(* Logix 5000 project; controller Safety vendor 1 type 14 code 86 rev 19.11; software revision 19.01; part 4 of 17 *)
(* tags used below, declared in another part *)
   A1_IO : UDT_CardSts[32];   // A1 Point I/O
   A1_IOSts_Flt : BOOL;   // A1 Point IO Module Fault ( 1= Faulted)
   A1_S20_ModFlt : ALIAS FOR Flt_Modules[0].0;   // A1 Point I/O Slot20 Module Fault (1 = Fault)
   A1_S21_ModFlt : ALIAS FOR Flt_Modules[0].1;   // A1 Point I/O Slot21 Module Fault (1 = Fault)
   C1_IO : UDT_CardSts[32];   // C1 Point I/O
   C1_IOSts_Flt : BOOL;   // C1 Point IO Module Fault ( 1= Faulted)
   C1_S12_ModFlt : ALIAS FOR Flt_Modules[0].2;   // C1 Point I/O Slot12 Module Fault (1 = Fault)
   ChgMe : BOOL;
   CHPLC_IO : UDT_CardSts[32];   // CHPLC Point I/O
   CHPLC_IOSts_Flt : BOOL;   // CHPLC Point IO Module Fault ( 1= Faulted)
   CHPLC_S1_ModFlt : ALIAS FOR Flt_Modules[0].3;   // CHPLC Point I/O Slot01 Module Fault (1 = Fault)
   CHPLC_S2_ModFlt : ALIAS FOR Flt_Modules[0].4;   // CHPLC Point I/O Slot02 Module Fault (1 = Fault)
   CHPLC_S3_ModFlt : ALIAS FOR Flt_Modules[0].5;   // CHPLC Point I/O Slot03 Module Fault (1 = Fault)
   CHPLC_S4_ModFlt : ALIAS FOR Flt_Modules[0].6;   // CHPLC Point I/O Slot04 Module Fault (1 = Fault)
   CHPLC_S5_ModFlt : ALIAS FOR Flt_Modules[0].7;   // CHPLC Point I/O Slot05 Module Fault (1 = Fault)
   CHPLC_S6_ModFlt : ALIAS FOR Flt_Modules[0].8;   // CHPLC Point I/O Slot06 Module Fault (1 = Fault)
   CommCards_OK : DINT;   // Comm Cards OK
   D1_IO : UDT_CardSts[32];   // D1 Point I/O
   D1_IOSts_Flt : BOOL;   // D1 Point IO Module Fault ( 1= Faulted)
   D1_S12_ModFlt : ALIAS FOR Flt_Modules[0].9;   // D1 Point I/O Slot12 Module Fault (1 = Fault)
   DPD_IO : UDT_CardSts[32];   // DPD Point I/O
   DPD_IOSts_Flt : BOOL;   // DPD Point IO Module Fault ( 1= Faulted)
   DPD_S14_ModFlt : ALIAS FOR Flt_Modules[0].10;   // DPD Point I/O Slot14 Module Fault (1 = Fault)
   DPD_S15_ModFlt : ALIAS FOR Flt_Modules[0].11;   // DPD Point I/O Slot15 Module Fault (1 = Fault)
   E1_IO : UDT_CardSts[32];   // E1 Point I/O
   E1_IOSts_Flt : BOOL;   // E1 Point IO Module Fault ( 1= Faulted)
   E1_S10_ModFlt : ALIAS FOR Flt_Modules[0].12;   // E1 Point I/O Slot10 Module Fault (1 = Fault)
   ES_IndJog_PB : BOOL;   // Exit Section Individual Jog Select ( 1= Req Individual)
   ES_Line_JogPB : BOOL;   // Exit Section Line Jog PB ( 1= Ind Jog )
   ES_Line_RunPB : BOOL;   // Exit Section Line Run PB ( 1= Run)
   ES_Line_StopPB : BOOL;   // Exit Section Line Stop PB ( 1= OK) (0=Stop)
   ES_Line_ThreadPB : BOOL;   // Exit Section Line Thread PB ( 1= Thread)
   ES_TndJog_PB : BOOL;   // Exit Section Tandem Jog PB (1= Tandem Jog Sel)
   ESTOP_x201PB040_Flt : ALIAS FOR Flt_Estops.0;   // OS1 Line EStop Pushbutton Fault ( 1= Fault)
   ESTOP_x211PB040_Flt : ALIAS FOR Flt_Estops.1;   // OS2 Line EStop Pushbutton Fault ( 1= Fault)
   ESTOP_x221PB040_Flt : ALIAS FOR Flt_Estops.2;   // OS3 Line EStop Pushbutton Fault ( 1= Fault)
   ESTOP_x231PB040_Flt : ALIAS FOR Flt_Estops.3;   // OS4N Line EStop Pushbutton Fault ( 1= Fault)
   ESTOP_x241PB040_Flt : ALIAS FOR Flt_Estops.4;   // OS4S Line EStop Pushbutton Fault ( 1= Fault)
   ESTOP_x251PB040_Flt : ALIAS FOR Flt_Estops.5;   // OS5 Line EStop Pushbutton Fault ( 1= Fault)
   ESTOP_x261PB040_Flt : ALIAS FOR Flt_Estops.6;   // OS6 Line EStop Pushbutton Fault ( 1= Fault)
   ESTOP_x271PB040_Flt : ALIAS FOR Flt_Estops.7;   // OS8 Line EStop Pushbutton Fault ( 1= Fault)
   ESTOP_x281PB040_Flt : ALIAS FOR Flt_Estops.8;   // OS9 Line EStop Pushbutton Fault ( 1= Fault)
   ESTOP_x291PB040_Flt : ALIAS FOR Flt_Estops.9;   // OS11 Line EStop Pushbutton Fault ( 1= Fault)
   ESTOP_x301PB040_Flt : ALIAS FOR Flt_Estops.10;   // OS13 Line EStop Pushbutton Fault ( 1= Fault)
   ESTOP_x311PB040_Flt : ALIAS FOR Flt_Estops.11;   // OS14 Line EStop Pushbutton Fault ( 1= Fault)
   ESTOP_x311PB130_Flt : ALIAS FOR Flt_Estops.17;   // OS14 Shear EStop Pushbutton Fault ( 1= Fault)
   ESTOP_x321PB040_Flt : ALIAS FOR Flt_Estops.12;   // OS15 Line EStop Pushbutton Fault ( 1= Fault)
   ESTOP_x331PB040_Flt : ALIAS FOR Flt_Estops.13;   // OS16 Line EStop Pushbutton Fault ( 1= Fault)
   ESTOP_x480PB470_Flt : ALIAS FOR Flt_Estops.14;   // DPD Line EStop Pushbutton Fault ( 1= Fault)
   ESTOP_x480PB550_Flt : ALIAS FOR Flt_Estops.15;   // DPD Line EStop Pushbutton Fault ( 1= Fault)
   ESTOP_x519LS470_Flt : ALIAS FOR Flt_Estops.18;   // G1 Line EStop Tripwire Limit Switch Fault ( 1= Fault)
   ESTOP_x533PB470_Flt : ALIAS FOR Flt_Estops.16;   // H1 Line EStop Pushbutton Fault ( 1= Fault)
   ExConHydPump_AutoStart : BOOL;   // (From Mach) Exit Conveyor Hydraulic Pump Auto Start Command
   F1_IO : UDT_CardSts[32];   // F1 Point I/O
   F1_IOSts_Flt : BOOL;   // F1 Point IO Module Fault ( 1= Faulted)
   F1_S19_ModFlt : ALIAS FOR Flt_Modules[0].13;   // F1 Point I/O Slot19 Module Fault (1 = Fault)
   F1_S20_ModFlt : ALIAS FOR Flt_Modules[0].14;   // F1 Point I/O Slot20 Module Fault (1 = Fault)
   Flt_Estops : DINT;   // Estop Fault Word
   Flt_Modules : DINT[5];   // Point IO Module Fault Word
   Flt_SafeOff : DINT[3];   // Safe Off Fault Word
   Flt_Starter : DINT;   // Starter Fault Word
   FltsToCitect : DINT[64];   // Faults to Citect
   FromCitect : DINT[64];   // (From Citect)
   FromMach : DINT[35];   // (FromMach)
   FromMachine : DINT[35];   // (FromMach)
   FromShearDie : DINT[35];   // (From Shear Die)
   FVR_y702MTR191_Flt : ALIAS FOR Flt_Starter.4;   // Rewind Pinch Roll Starter Fault ( 1= Fault)
   FVR_y708MTR080_Flt : ALIAS FOR Flt_Starter.1;   // Flattener Drive Motor Starter Fault ( 1= Fault)
   FVR_y708MTR250_Flt : ALIAS FOR Flt_Starter.0;   // Unwind Hold Down Roll Starter Fault ( 1= Fault)
   FVR_y753MTR190_Flt : ALIAS FOR Flt_Starter.2;   // Trimmer Pinch Roll Starter Fault ( 1= Fault)
   FVR_y761MTR081_Flt : ALIAS FOR Flt_Starter.3;   // Trimmer Scrap Conveyor Starter Fault ( 1= Fault)
   FVR_y778MTR080_Flt : ALIAS FOR Flt_Starter.5;   // Shear Die Crank Starter Fault ( 1= Fault)
   FVR_y802MTR080_Flt : ALIAS FOR Flt_Starter.6;   // Stacker Side Guide Lift Starter Fault ( 1= Fault)
   FVR_y802MTR230_Flt : ALIAS FOR Flt_Starter.8;   // Scrap Horizontal Conveyor Starter Fault ( 1= Fault)
   FVR_y802MTR231_Flt : ALIAS FOR Flt_Starter.7;   // Stacker Chain Conveyor Starter Fault ( 1= Fault)
   G1_IO : UDT_CardSts[32];   // G1 Point I/O
   G1_IOSts_Flt : BOOL;   // G1 Point IO Module Fault ( 1= Faulted)
   G1_S11_ModFlt : ALIAS FOR Flt_Modules[0].15;   // G1 Point I/O Slot11 Module Fault (1 = Fault)
   G1_S12_ModFlt : ALIAS FOR Flt_Modules[0].16;   // G1 Point I/O Slot12 Module Fault (1 = Fault)
   H1_IO : UDT_CardSts[32];   // H1 Point I/O
   H1_IOSts_Flt : BOOL;   // H1 Point IO Module Fault ( 1= Faulted)
   H1_S5_ModFlt : ALIAS FOR Flt_Modules[0].17;   // H1 Point I/O Slot05 Module Fault (1 = Fault)
   H1_S6_ModFlt : ALIAS FOR Flt_Modules[0].18;   // H1 Point I/O Slot06 Module Fault (1 = Fault)
   HydPumps_AutoStart : BOOL;   // (From Mach) Hydraulic Pumps Auto Start Active
   IOCards_OK : DINT;   // Point I/O Cards OK
   Local_ModFlts : DINT;   // Local Card Fault Status
   LubePumps_AutoStart : BOOL;   // (From Mach) Lube Pumps Auto Start Active
   Machine_HB_Flt : BOOL;   // Machine Heartbeat Fault ( 1= Fault)
   MCC1_IO : UDT_CardSts[32];   // MCC1 Point I/O
   MCC1_IOSts_Flt : BOOL;   // MCC1 Point IO Module Fault ( 1= Faulted)
   MCC1_S1_ModFlt : ALIAS FOR Flt_Modules[2].0;   // MCC1 Point I/O Slot01 Module Fault (1 = Fault)
   MCC1_S6_ModFlt : ALIAS FOR Flt_Modules[2].1;   // MCC1 Point I/O Slot06 Module Fault (1 = Fault)
   MCC2_IO : UDT_CardSts[32];   // MCC2 Point I/O
   MCC2_IOSts_Flt : BOOL;   // MCC2 Point IO Module Fault ( 1= Faulted)
   MCC2_S1_ModFlt : ALIAS FOR Flt_Modules[2].2;   // MCC2 Point I/O Slot01 Module Fault (1 = Fault)
   MCC2_S2_ModFlt : ALIAS FOR Flt_Modules[2].3;   // MCC2 Point I/O Slot02 Module Fault (1 = Fault)
   MCC3_IO : UDT_CardSts[32];   // MCC3 Point I/O
   MCC3_IOSts_Flt : BOOL;   // MCC3 Point IO Module Fault ( 1= Faulted)
   MCC3_S1_ModFlt : ALIAS FOR Flt_Modules[2].4;   // MCC3 Point I/O Slot01 Module Fault (1 = Fault)
   MCC3_S3_ModFlt : ALIAS FOR Flt_Modules[2].5;   // MCC3 Point I/O Slot03 Module Fault (1 = Fault)
   MCC3_S4_ModFlt : ALIAS FOR Flt_Modules[2].6;   // MCC3 Point I/O Slot04 Module Fault (1 = Fault)
   MCC4_IO : UDT_CardSts[32];   // MCC4 Point I/O
   MCC4_IOSts_Flt : BOOL;   // MCC-4 Point IO Module Fault ( 1= Faulted)
   MCC4_S1_ModFlt : ALIAS FOR Flt_Modules[2].7;   // MCC4 Point I/O Slot01 Module Fault (1 = Fault)
   MCC4_S3_ModFlt : ALIAS FOR Flt_Modules[2].8;   // MCC4 Point I/O Slot03 Module Fault (1 = Fault)
   MCC4_S4_ModFlt : ALIAS FOR Flt_Modules[2].9;   // MCC4 Point I/O Slot04 Module Fault (1 = Fault)
   MCC5_IO : UDT_CardSts[32];   // MCC5 Point I/O
   MCC5_IOSts_Flt : BOOL;   // MCC-5 Point IO Module Fault ( 1= Faulted)
   MCC5_S1_ModFlt : ALIAS FOR Flt_Modules[2].10;   // MCC5 Point I/O Slot01 Module Fault (1 = Fault)
   MCC5_S3_ModFlt : ALIAS FOR Flt_Modules[2].11;   // MCC5 Point I/O Slot03 Module Fault (1 = Fault)
   MCC5_S4_ModFlt : ALIAS FOR Flt_Modules[2].12;   // MCC5 Point I/O Slot04 Module Fault (1 = Fault)
   MCC5_S5_ModFlt : ALIAS FOR Flt_Modules[2].13;   // MCC5 Point I/O Slot05 Module Fault (1 = Fault)
   OS11_IO : UDT_CardSts[32];   // OS11 Point I/O
   OS11_IOSts_Flt : BOOL;   // OS11 Point IO Module Fault ( 1= Faulted)
   OS11_S1_ModFlt : ALIAS FOR Flt_Modules[1].11;   // OS11 Point I/O Slot01 Module Fault (1 = Fault)
   OS13_IO : UDT_CardSts[32];   // OS13 Point I/O
   OS13_IOSts_Flt : BOOL;   // OS13 Point IO Module Fault ( 1= Faulted)
   OS13_S1_ModFlt : ALIAS FOR Flt_Modules[1].12;   // OS13 Point I/O Slot01 Module Fault (1 = Fault)
   OS14_IO : UDT_CardSts[32];   // OS14 Point I/O
   OS14_IOSts_Flt : BOOL;   // OS14 Point IO Module Fault ( 1= Faulted)
   OS14_S1_ModFlt : ALIAS FOR Flt_Modules[1].13;   // OS14 Point I/O Slot01 Module Fault (1 = Fault)
   OS15_IO : UDT_CardSts[32];   // OS15 Point I/O
   OS15_IOSts_Flt : BOOL;   // OS15 Point IO Module Fault ( 1= Faulted)
   OS15_S1_ModFlt : ALIAS FOR Flt_Modules[1].14;   // OS15 Point I/O Slot01 Module Fault (1 = Fault)
   OS16_IO : UDT_CardSts[32];   // OS16 Point I/O
   OS16_IOSts_Flt : BOOL;   // OS16 Point IO Module Fault ( 1= Faulted)
   OS16_S1_ModFlt : ALIAS FOR Flt_Modules[1].15;   // OS16 Point I/O Slot01 Module Fault (1 = Fault)
   OS1_IO : UDT_CardSts[32];   // OS1 Point I/O
   OS1_IOSts_Flt : BOOL;   // OS1 Point IO Module Fault ( 1= Faulted)
   OS1_S1_ModFlt : ALIAS FOR Flt_Modules[1].0;   // OS1 Point I/O Slot01 Module Fault (1 = Fault)
   OS2_IO : UDT_CardSts[32];   // OS2 Point I/O
   OS2_IOSts_Flt : BOOL;   // OS2 Point IO Module Fault ( 1= Faulted)
   OS2_S1_ModFlt : ALIAS FOR Flt_Modules[1].1;   // OS2 Point I/O Slot01 Module Fault (1 = Fault)
   OS3_IO : UDT_CardSts[32];   // OS3 Point I/O
   OS3_IOSts_Flt : BOOL;   // OS3 Point IO Module Fault ( 1= Faulted)
   OS3_S1_ModFlt : ALIAS FOR Flt_Modules[1].2;   // OS3 Point I/O Slot01 Module Fault (1 = Fault)
   OS4N_IO : UDT_CardSts[32];   // OS4N Point I/O
   OS4N_IOSts_Flt : BOOL;   // OS4N Point IO Module Fault ( 1= Faulted)
   OS4N_S1_ModFlt : ALIAS FOR Flt_Modules[1].3;   // OS4N Point I/O Slot01 Module Fault (1 = Fault)
   OS4N_S5_ModFlt : ALIAS FOR Flt_Modules[1].4;   // OS4N Point I/O Slot05 Module Fault (1 = Fault)
   OS4S_IO : UDT_CardSts[32];   // OS4S Point I/O
   OS4S_IOSts_Flt : BOOL;   // OS4S Point IO Module Fault ( 1= Faulted)
   OS4S_S1_ModFlt : ALIAS FOR Flt_Modules[1].5;   // OS4S Point I/O Slot01 Module Fault (1 = Fault)
   OS4S_S5_ModFlt : ALIAS FOR Flt_Modules[1].6;   // OS4S Point I/O Slot05 Module Fault (1 = Fault)
   OS5_IO : UDT_CardSts[32];   // OS5 Point I/O
   OS5_IOSts_Flt : BOOL;   // OS5 Point IO Module Fault ( 1= Faulted)
   OS5_S1_ModFlt : ALIAS FOR Flt_Modules[1].7;   // OS5 Point I/O Slot01 Module Fault (1 = Fault)
   OS6_IO : UDT_CardSts[32];   // OS6 Point I/O
   OS6_IOSts_Flt : BOOL;   // OS6 Point IO Module Fault ( 1= Faulted)
   OS6_S1_ModFlt : ALIAS FOR Flt_Modules[1].8;   // OS6 Point I/O Slot01 Module Fault (1 = Fault)
   OS8_IO : UDT_CardSts[32];   // OS8 Point I/O
   OS8_IOSts_Flt : BOOL;   // OS8 Point IO Module Fault ( 1= Faulted)
   OS8_S1_ModFlt : ALIAS FOR Flt_Modules[1].9;   // OS8 Point I/O Slot01 Module Fault (1 = Fault)
   OS9_IO : UDT_CardSts[32];   // OS9 Point I/O
   OS9_IOSts_Flt : BOOL;   // OS9 Point IO Module Fault ( 1= Faulted)
   OS9_S1_ModFlt : ALIAS FOR Flt_Modules[1].10;   // OS9 Point I/O Slot01 Module Fault (1 = Fault)
   Rem_ModFlts : DINT;   // Remote IO Comm Faults
   SafeOff_y172CR460_Flt : ALIAS FOR Flt_SafeOff[0].0;   // Shear Die Main Contactor Relay Fault ( 1= Fault)
   SafeOff_y172CR510_Flt : ALIAS FOR Flt_SafeOff[0].1;   // Shear Die Drive Enable Relay Fault ( 1= Fault)
   SafeOff_y613CR460_Flt : ALIAS FOR Flt_SafeOff[0].2;   // Unwind Op Side Main Contactor Relay Fault ( 1= Fault)
   SafeOff_y613CR510_Flt : ALIAS FOR Flt_SafeOff[0].3;   // Unwind Op Side Drive Enable Relay Fault ( 1= Fault)
   SafeOff_y613CR550_Flt : ALIAS FOR Flt_SafeOff[0].4;   // Unwind Drive Side Main Contactor Relay Fault ( 1= Fault)
   SafeOff_y613CR590_Flt : ALIAS FOR Flt_SafeOff[0].5;   // Unwind Drive Side Drive Enable Relay Fault ( 1= Fault)
   SafeOff_y613CR630_Flt : ALIAS FOR Flt_SafeOff[0].6;   // #1 Entry Bridle Roll 2 Main Contactor Relay Fault ( 1= Fault)
   SafeOff_y613CR670_Flt : ALIAS FOR Flt_SafeOff[0].7;   // #1 Entry Bridle Roll 2 Drive Enable Relay Fault ( 1= Fault)
   SafeOff_y613CR710_Flt : ALIAS FOR Flt_SafeOff[0].8;   // #2 Entry Bridle Roll 3 Main Contactor Relay Fault ( 1= Fault)
   SafeOff_y613CR750_Flt : ALIAS FOR Flt_SafeOff[0].9;   // #2 Entry Bridle Roll 3 Drive Enable Relay Fault ( 1= Fault)
   SafeOff_y614CR040_Flt : ALIAS FOR Flt_SafeOff[0].10;   // #1 Exit Bridle Roll 6 Main Contactor Relay Fault ( 1= Fault)
   SafeOff_y614CR090_Flt : ALIAS FOR Flt_SafeOff[0].11;   // #1 Exit Bridle Roll 6 Drive Enable Relay Fault ( 1= Fault)
   SafeOff_y614CR130_Flt : ALIAS FOR Flt_SafeOff[0].12;   // #2 Exit Bridle Roll 7 Main Contactor Relay Fault ( 1= Fault)
   SafeOff_y614CR170_Flt : ALIAS FOR Flt_SafeOff[0].13;   // #2 Exit Bridle Roll 7 Drive Enable Relay Fault ( 1= Fault)
   SafeOff_y614CR210_Flt : ALIAS FOR Flt_SafeOff[0].14;   // Rewind Main Contactor Relay Fault ( 1= Fault)
   SafeOff_y614CR250_Flt : ALIAS FOR Flt_SafeOff[0].15;   // Rewind Drive Enable Relay Fault ( 1= Fault)
   ScrapModeOn : BOOL;   // Scrap Mode Selected ( 1= Requested)
   SDPLC_IO : UDT_CardSts[32];   // SDPLC Point I/O
   SDPLC_IOSts_Flt : BOOL;   // SDPLC Point IO Module Fault ( 1= Faulted)
   SDPLC_S1_ModFlt : ALIAS FOR Flt_Modules[0].19;   // SDPLC Point I/O Slot01 Module Fault (1 = Fault)
   SDPLC_S2_ModFlt : ALIAS FOR Flt_Modules[0].20;   // SDPLC Point I/O Slot02 Module Fault (1 = Fault)
   Shear_HB_Flt : BOOL;   // Shear Heartbeat Fault ( 1= Fault)
   SrPRLubePump_AutoStart : BOOL;   // (From Mach) Shear Pinch Roll Lube Pump Auto Start Command
   StHydPump_AutoStart : BOOL;   // (From Mach) Sheeter Hydraulic Pump Auto Start Command
   StPRLubePump_AutoStart : BOOL;   // (From Mach) Sheeter Pinch Roll Lube Pump Auto Start Command
   Sy_ClrFlt : BOOL;   // System Clear Fault
   VS2_IO : UDT_CardSts[32];   // VS2 Point I/O
   VS2_IOSts_Flt : BOOL;   // VS2 Point IO Module Fault ( 1= Faulted)
   VS2_S10_ModFlt : ALIAS FOR Flt_Modules[0].21;   // VS2 Point I/O Slot10 Module Fault (1 = Fault)
   x301SS540a : BOOL;   // Sheeter Pinch Roll Jog Forward SS
   x301SS540b : BOOL;   // Sheeter Pinch Roll Jog Reverse SS
   x312PB700 : BOOL;   // Product Conveyor Jog Forward PB
   x312PB740 : BOOL;   // Product Conveyor Jog Reverse PB
   x312SS460a : BOOL;   // Scrap Conveyor Jog Forward SS
   x312SS460b : BOOL;   // Scrap Conveyor Jog Reverse SS
   x313SS460a : BOOL;   // Shear Conveyor Jog Forward SS
   x313SS460b : BOOL;   // Shear Conveyor Jog Reverse SS
   x314SS040a : BOOL;   // Shear Pinch Roll Jog Forward SS
   x314SS040b : BOOL;   // Shear Pinch Roll Jog Reverse SS
   x315SS040a : BOOL;   // Sheeter Pinch Roll Jog Forward SS
   x315SS040b : BOOL;   // Sheeter Pinch Roll Jog Reverse SS
   x775MTR280RF : BOOL;   // (From Shear DIe) Shear Pinch Roll Lube Run Fdbk
   x781MTR080RF : BOOL;   // (From Shear DIe) Sheeter Pinch Roll Lube Run Fdbk
   x781MTR190RF : BOOL;   // (From Shear DIe) Sheeter Hyd Pump Run Fdbk
   x813MTR080RF : BOOL;   // (From Shear DIe) Exit Conveyor Hyd Pump Run Fdbk
(* CardSts, continued *)

ROUTINE Remote_IO   (* ladder *)
// Remote IO Card Status
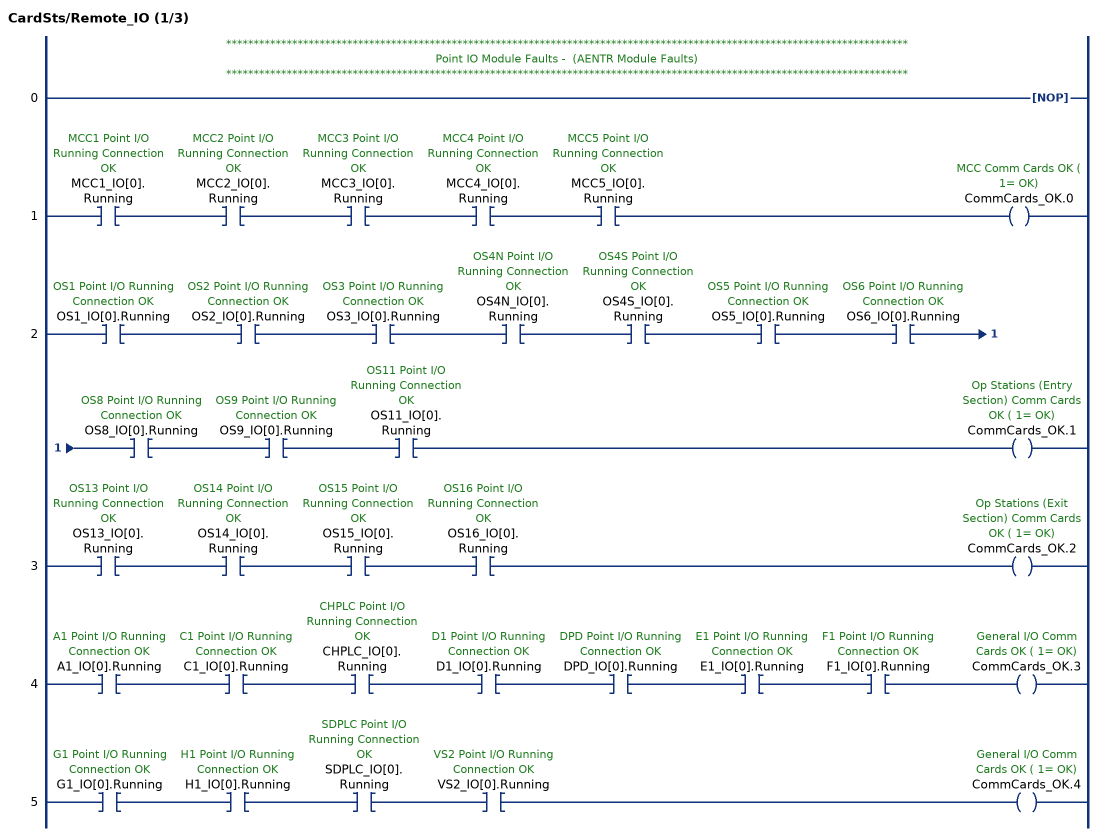
   // ****************************************************************************************************************************
   // Point IO Module Faults -  (AENTR Module Faults)
   // ****************************************************************************************************************************
   0: NOP();
   1: XIC(MCC1_IO[0].Running)XIC(MCC2_IO[0].Running)XIC(MCC3_IO[0].Running)XIC(MCC4_IO[0].Running)XIC(MCC5_IO[0].Running)OTE(CommCards_OK.0);
   2: XIC(OS1_IO[0].Running)XIC(OS2_IO[0].Running)XIC(OS3_IO[0].Running)XIC(OS4N_IO[0].Running)XIC(OS4S_IO[0].Running)XIC(OS5_IO[0].Running)XIC(OS6_IO[0].Running)XIC(OS8_IO[0].Running)XIC(OS9_IO[0].Running)XIC(OS11_IO[0].Running)OTE(CommCards_OK.1);
   3: XIC(OS13_IO[0].Running)XIC(OS14_IO[0].Running)XIC(OS15_IO[0].Running)XIC(OS16_IO[0].Running)OTE(CommCards_OK.2);
   4: XIC(A1_IO[0].Running)XIC(C1_IO[0].Running)XIC(CHPLC_IO[0].Running)XIC(D1_IO[0].Running)XIC(DPD_IO[0].Running)XIC(E1_IO[0].Running)XIC(F1_IO[0].Running)OTE(CommCards_OK.3);
   5: XIC(G1_IO[0].Running)XIC(H1_IO[0].Running)XIC(SDPLC_IO[0].Running)XIC(VS2_IO[0].Running)OTE(CommCards_OK.4);
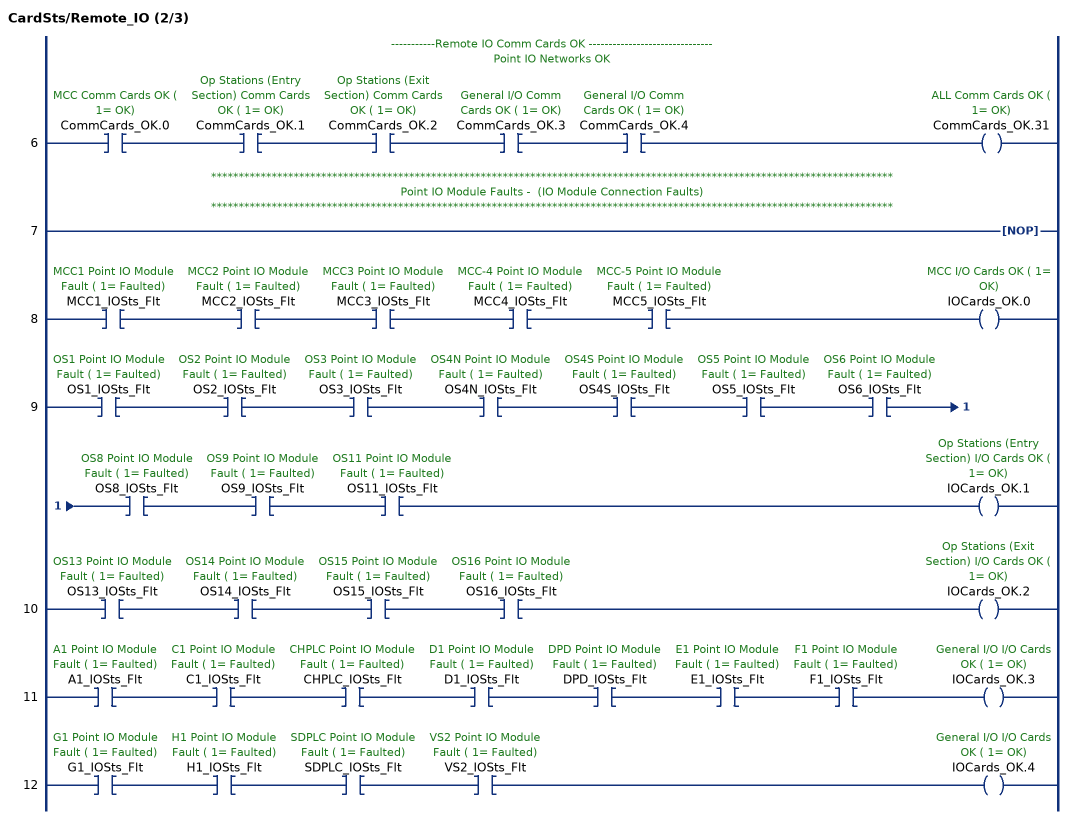
   // -----------Remote IO Comm Cards OK -------------------------------
   // Point IO Networks OK
   6: XIC(CommCards_OK.0)XIC(CommCards_OK.1)XIC(CommCards_OK.2)XIC(CommCards_OK.3)XIC(CommCards_OK.4)OTE(CommCards_OK.31);
   // ****************************************************************************************************************************
   // Point IO Module Faults -  (IO Module Connection Faults)
   // ****************************************************************************************************************************
   7: NOP();
   8: XIC(MCC1_IOSts_Flt)XIC(MCC2_IOSts_Flt)XIC(MCC3_IOSts_Flt)XIC(MCC4_IOSts_Flt)XIC(MCC5_IOSts_Flt)OTE(IOCards_OK.0);
   9: XIC(OS1_IOSts_Flt)XIC(OS2_IOSts_Flt)XIC(OS3_IOSts_Flt)XIC(OS4N_IOSts_Flt)XIC(OS4S_IOSts_Flt)XIC(OS5_IOSts_Flt)XIC(OS6_IOSts_Flt)XIC(OS8_IOSts_Flt)XIC(OS9_IOSts_Flt)XIC(OS11_IOSts_Flt)OTE(IOCards_OK.1);
   10: XIC(OS13_IOSts_Flt)XIC(OS14_IOSts_Flt)XIC(OS15_IOSts_Flt)XIC(OS16_IOSts_Flt)OTE(IOCards_OK.2);
   11: XIC(A1_IOSts_Flt)XIC(C1_IOSts_Flt)XIC(CHPLC_IOSts_Flt)XIC(D1_IOSts_Flt)XIC(DPD_IOSts_Flt)XIC(E1_IOSts_Flt)XIC(F1_IOSts_Flt)OTE(IOCards_OK.3);
   12: XIC(G1_IOSts_Flt)XIC(H1_IOSts_Flt)XIC(SDPLC_IOSts_Flt)XIC(VS2_IOSts_Flt)OTE(IOCards_OK.4);
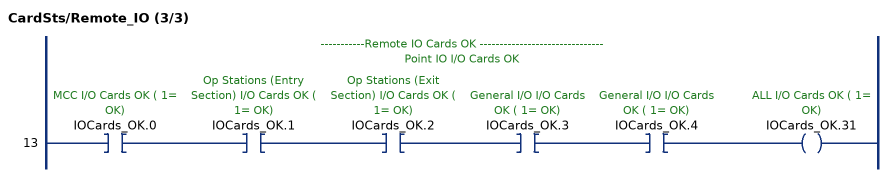
   // -----------Remote IO Cards OK -------------------------------
   // Point IO I/O Cards OK
   13: XIC(IOCards_OK.0)XIC(IOCards_OK.1)XIC(IOCards_OK.2)XIC(IOCards_OK.3)XIC(IOCards_OK.4)OTE(IOCards_OK.31);
END_ROUTINE

ROUTINE SDPLC_IO   (* ladder *)
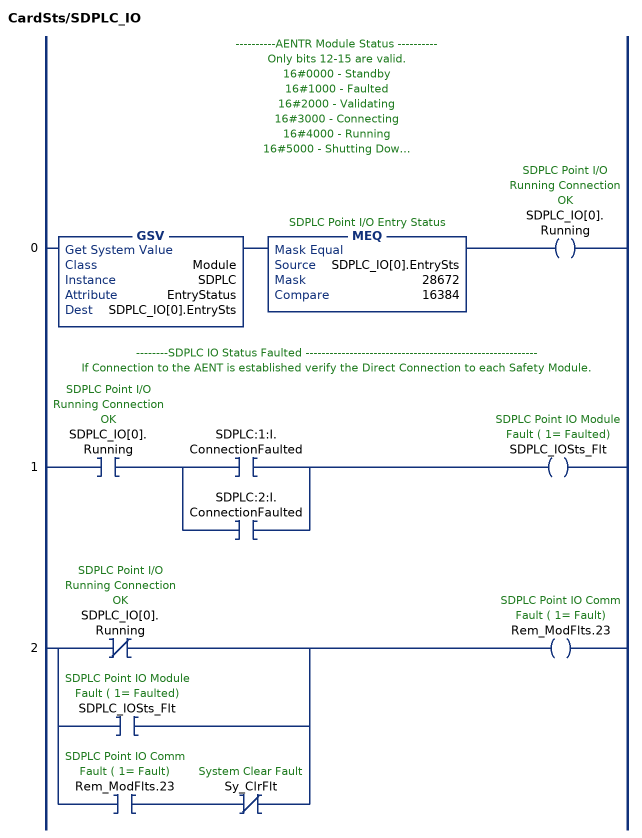
   // ----------AENTR Module Status ----------
   // Only bits 12-15 are valid.
   // 16#0000 - Standby
   // 16#1000 - Faulted
   // 16#2000 - Validating
   // 16#3000 - Connecting
   // 16#4000 - Running
   // 16#5000 - Shutting Down
   // 16#6000 - Inhibited
   // 16#7000 - Waiting
   0: GSV(Module,SDPLC,EntryStatus,SDPLC_IO[0].EntrySts)MEQ(SDPLC_IO[0].EntrySts,28672,16384)OTE(SDPLC_IO[0].Running);
   // --------SDPLC IO Status Faulted ----------------------------------------------------------
   // If Connection to the AENT is established verify the Direct Connection to each Safety Module.
   1: XIC(SDPLC_IO[0].Running)[XIC(SDPLC:1:I.ConnectionFaulted) ,XIC(SDPLC:2:I.ConnectionFaulted) ]OTE(SDPLC_IOSts_Flt);
   2: [XIO(SDPLC_IO[0].Running) ,XIC(SDPLC_IOSts_Flt) ,XIC(Rem_ModFlts.23) XIO(Sy_ClrFlt) ]OTE(Rem_ModFlts.23);
END_ROUTINE

ROUTINE VS2_IO   (* ladder *)
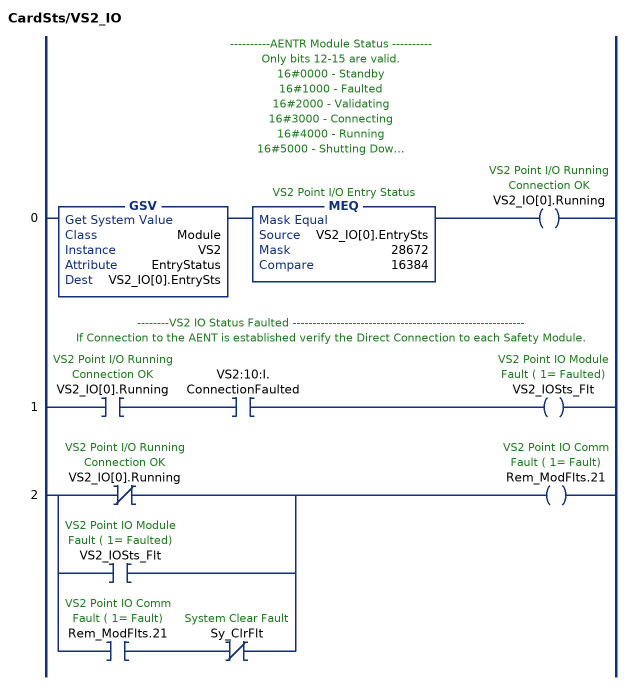
   // ----------AENTR Module Status ----------
   // Only bits 12-15 are valid.
   // 16#0000 - Standby
   // 16#1000 - Faulted
   // 16#2000 - Validating
   // 16#3000 - Connecting
   // 16#4000 - Running
   // 16#5000 - Shutting Down
   // 16#6000 - Inhibited
   // 16#7000 - Waiting
   0: GSV(Module,VS2,EntryStatus,VS2_IO[0].EntrySts)MEQ(VS2_IO[0].EntrySts,28672,16384)OTE(VS2_IO[0].Running);
   // --------VS2 IO Status Faulted ----------------------------------------------------------
   // If Connection to the AENT is established verify the Direct Connection to each Safety Module.
   1: XIC(VS2_IO[0].Running)XIC(VS2:10:I.ConnectionFaulted)OTE(VS2_IOSts_Flt);
   2: [XIO(VS2_IO[0].Running) ,XIC(VS2_IOSts_Flt) ,XIC(Rem_ModFlts.21) XIO(Sy_ClrFlt) ]OTE(Rem_ModFlts.21);
END_ROUTINE
END_PROGRAM

PROGRAM Comms   (* main routine MainRoutine *)
// Communications to Others

ROUTINE FltsToCitect   (* ladder *)
// Faults to the
// Citect System
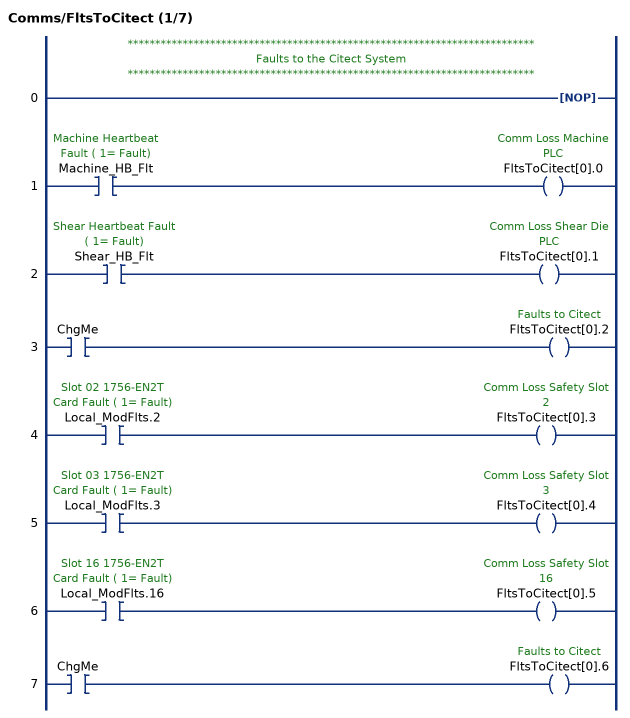
   // **************************************************************************
   // Faults to the Citect System
   // **************************************************************************
   0: NOP();
   1: XIC(Machine_HB_Flt)OTE(FltsToCitect[0].0);
   2: XIC(Shear_HB_Flt)OTE(FltsToCitect[0].1);
   3: XIC(ChgMe)OTE(FltsToCitect[0].2);
   4: XIC(Local_ModFlts.2)OTE(FltsToCitect[0].3);
   5: XIC(Local_ModFlts.3)OTE(FltsToCitect[0].4);
   6: XIC(Local_ModFlts.16)OTE(FltsToCitect[0].5);
   7: XIC(ChgMe)OTE(FltsToCitect[0].6);
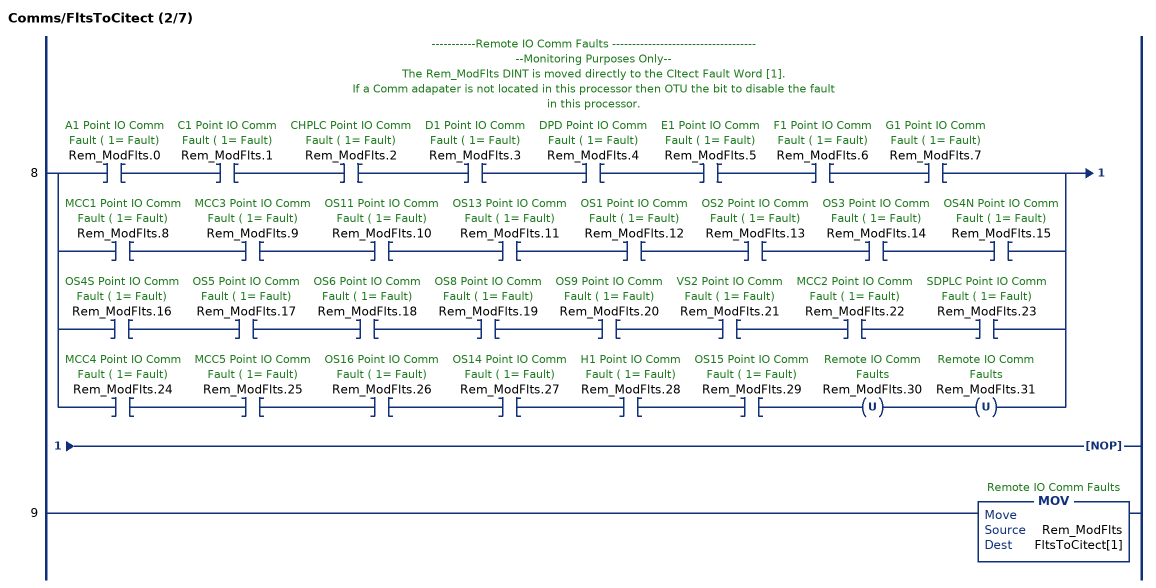
   // -----------Remote IO Comm Faults ------------------------------------
   // --Monitoring Purposes Only--
   // The Rem_ModFlts DINT is moved directly to the CItect Fault Word [1].
   // If a Comm adapater is not located in this processor then OTU the bit to disable the fault
   // in this processor.
   8: [XIC(Rem_ModFlts.0) XIC(Rem_ModFlts.1) XIC(Rem_ModFlts.2) XIC(Rem_ModFlts.3) XIC(Rem_ModFlts.4) XIC(Rem_ModFlts.5) XIC(Rem_ModFlts.6) XIC(Rem_ModFlts.7) ,XIC(Rem_ModFlts.8) XIC(Rem_ModFlts.9) XIC(Rem_ModFlts.10) XIC(Rem_ModFlts.11) XIC(Rem_ModFlts.12) XIC(Rem_ModFlts.13) XIC(Rem_ModFlts.14) XIC(Rem_ModFlts.15) ,XIC(Rem_ModFlts.16) XIC(Rem_ModFlts.17) XIC(Rem_ModFlts.18) XIC(Rem_ModFlts.19) XIC(Rem_ModFlts.20) XIC(Rem_ModFlts.21) XIC(Rem_ModFlts.22) XIC(Rem_ModFlts.23) ,XIC(Rem_ModFlts.24) XIC(Rem_ModFlts.25) XIC(Rem_ModFlts.26) XIC(Rem_ModFlts.27) XIC(Rem_ModFlts.28) XIC(Rem_ModFlts.29) OTU(Rem_ModFlts.30) OTU(Rem_ModFlts.31) ]NOP();
   9: MOV(Rem_ModFlts,FltsToCitect[1]);
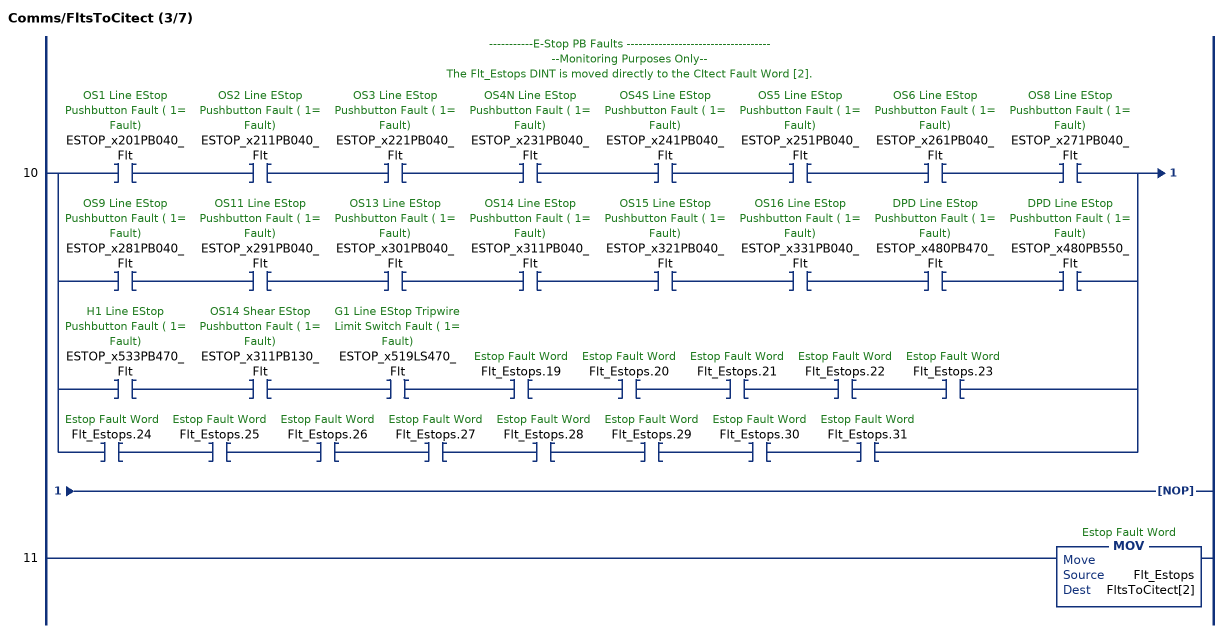
   // -----------E-Stop PB Faults ------------------------------------
   // --Monitoring Purposes Only--
   // The Flt_Estops DINT is moved directly to the CItect Fault Word [2].
   10: [XIC(ESTOP_x201PB040_Flt) XIC(ESTOP_x211PB040_Flt) XIC(ESTOP_x221PB040_Flt) XIC(ESTOP_x231PB040_Flt) XIC(ESTOP_x241PB040_Flt) XIC(ESTOP_x251PB040_Flt) XIC(ESTOP_x261PB040_Flt) XIC(ESTOP_x271PB040_Flt) ,XIC(ESTOP_x281PB040_Flt) XIC(ESTOP_x291PB040_Flt) XIC(ESTOP_x301PB040_Flt) XIC(ESTOP_x311PB040_Flt) XIC(ESTOP_x321PB040_Flt) XIC(ESTOP_x331PB040_Flt) XIC(ESTOP_x480PB470_Flt) XIC(ESTOP_x480PB550_Flt) ,XIC(ESTOP_x533PB470_Flt) XIC(ESTOP_x311PB130_Flt) XIC(ESTOP_x519LS470_Flt) XIC(Flt_Estops.19) XIC(Flt_Estops.20) XIC(Flt_Estops.21) XIC(Flt_Estops.22) XIC(Flt_Estops.23) ,XIC(Flt_Estops.24) XIC(Flt_Estops.25) XIC(Flt_Estops.26) XIC(Flt_Estops.27) XIC(Flt_Estops.28) XIC(Flt_Estops.29) XIC(Flt_Estops.30) XIC(Flt_Estops.31) ]NOP();
   11: MOV(Flt_Estops,FltsToCitect[2]);
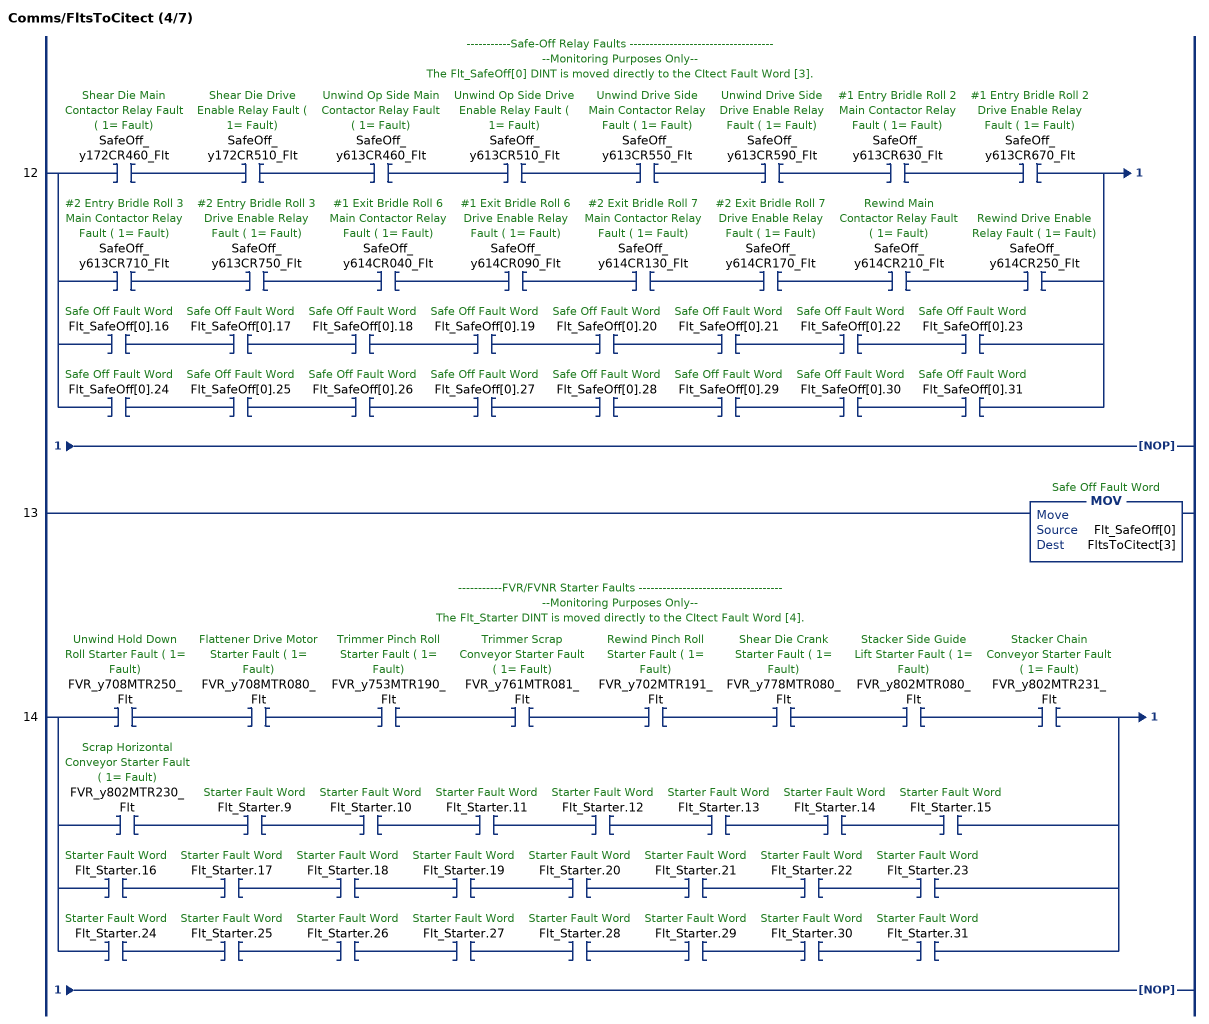
   // -----------Safe-Off Relay Faults ------------------------------------
   // --Monitoring Purposes Only--
   // The Flt_SafeOff[0] DINT is moved directly to the CItect Fault Word [3].
   12: [XIC(SafeOff_y172CR460_Flt) XIC(SafeOff_y172CR510_Flt) XIC(SafeOff_y613CR460_Flt) XIC(SafeOff_y613CR510_Flt) XIC(SafeOff_y613CR550_Flt) XIC(SafeOff_y613CR590_Flt) XIC(SafeOff_y613CR630_Flt) XIC(SafeOff_y613CR670_Flt) ,XIC(SafeOff_y613CR710_Flt) XIC(SafeOff_y613CR750_Flt) XIC(SafeOff_y614CR040_Flt) XIC(SafeOff_y614CR090_Flt) XIC(SafeOff_y614CR130_Flt) XIC(SafeOff_y614CR170_Flt) XIC(SafeOff_y614CR210_Flt) XIC(SafeOff_y614CR250_Flt) ,XIC(Flt_SafeOff[0].16) XIC(Flt_SafeOff[0].17) XIC(Flt_SafeOff[0].18) XIC(Flt_SafeOff[0].19) XIC(Flt_SafeOff[0].20) XIC(Flt_SafeOff[0].21) XIC(Flt_SafeOff[0].22) XIC(Flt_SafeOff[0].23) ,XIC(Flt_SafeOff[0].24) XIC(Flt_SafeOff[0].25) XIC(Flt_SafeOff[0].26) XIC(Flt_SafeOff[0].27) XIC(Flt_SafeOff[0].28) XIC(Flt_SafeOff[0].29) XIC(Flt_SafeOff[0].30) XIC(Flt_SafeOff[0].31) ]NOP();
   13: MOV(Flt_SafeOff[0],FltsToCitect[3]);
   // -----------FVR/FVNR Starter Faults ------------------------------------
   // --Monitoring Purposes Only--
   // The Flt_Starter DINT is moved directly to the CItect Fault Word [4].
   14: [XIC(FVR_y708MTR250_Flt) XIC(FVR_y708MTR080_Flt) XIC(FVR_y753MTR190_Flt) XIC(FVR_y761MTR081_Flt) XIC(FVR_y702MTR191_Flt) XIC(FVR_y778MTR080_Flt) XIC(FVR_y802MTR080_Flt) XIC(FVR_y802MTR231_Flt) ,XIC(FVR_y802MTR230_Flt) XIC(Flt_Starter.9) XIC(Flt_Starter.10) XIC(Flt_Starter.11) XIC(Flt_Starter.12) XIC(Flt_Starter.13) XIC(Flt_Starter.14) XIC(Flt_Starter.15) ,XIC(Flt_Starter.16) XIC(Flt_Starter.17) XIC(Flt_Starter.18) XIC(Flt_Starter.19) XIC(Flt_Starter.20) XIC(Flt_Starter.21) XIC(Flt_Starter.22) XIC(Flt_Starter.23) ,XIC(Flt_Starter.24) XIC(Flt_Starter.25) XIC(Flt_Starter.26) XIC(Flt_Starter.27) XIC(Flt_Starter.28) XIC(Flt_Starter.29) XIC(Flt_Starter.30) XIC(Flt_Starter.31) ]NOP();
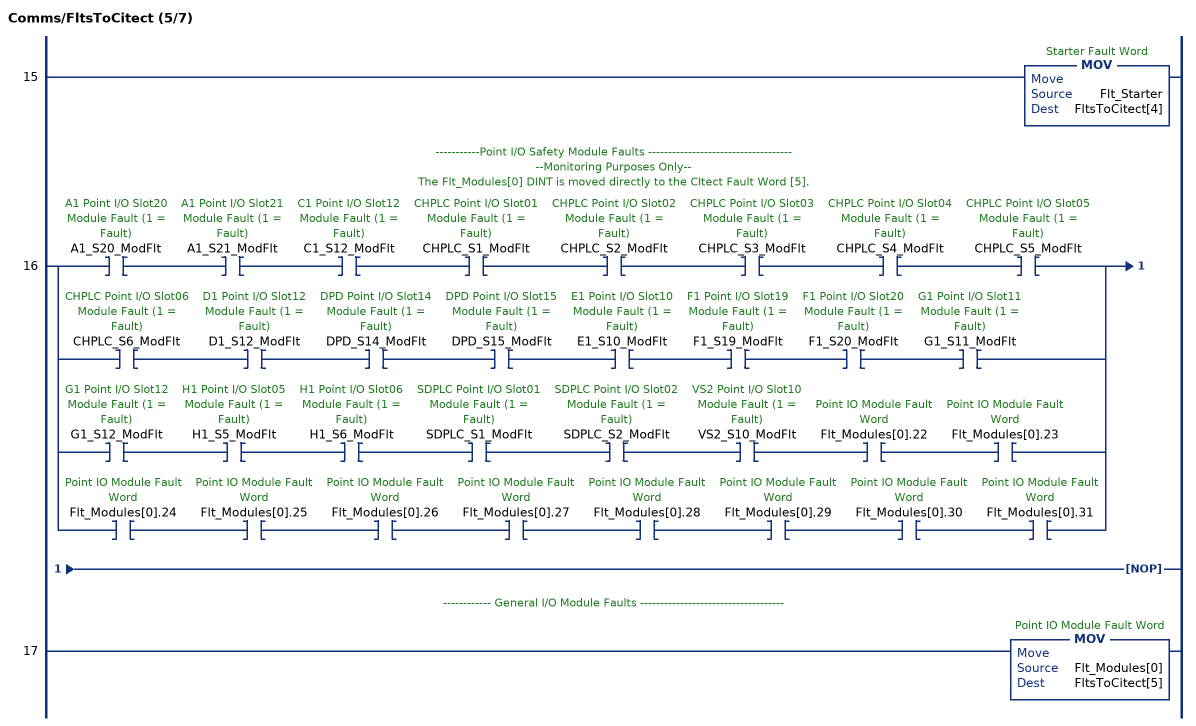
   15: MOV(Flt_Starter,FltsToCitect[4]);
   // -----------Point I/O Safety Module Faults ------------------------------------
   // --Monitoring Purposes Only--
   // The Flt_Modules[0] DINT is moved directly to the CItect Fault Word [5].
   16: [XIC(A1_S20_ModFlt) XIC(A1_S21_ModFlt) XIC(C1_S12_ModFlt) XIC(CHPLC_S1_ModFlt) XIC(CHPLC_S2_ModFlt) XIC(CHPLC_S3_ModFlt) XIC(CHPLC_S4_ModFlt) XIC(CHPLC_S5_ModFlt) ,XIC(CHPLC_S6_ModFlt) XIC(D1_S12_ModFlt) XIC(DPD_S14_ModFlt) XIC(DPD_S15_ModFlt) XIC(E1_S10_ModFlt) XIC(F1_S19_ModFlt) XIC(F1_S20_ModFlt) XIC(G1_S11_ModFlt) ,XIC(G1_S12_ModFlt) XIC(H1_S5_ModFlt) XIC(H1_S6_ModFlt) XIC(SDPLC_S1_ModFlt) XIC(SDPLC_S2_ModFlt) XIC(VS2_S10_ModFlt) XIC(Flt_Modules[0].22) XIC(Flt_Modules[0].23) ,XIC(Flt_Modules[0].24) XIC(Flt_Modules[0].25) XIC(Flt_Modules[0].26) XIC(Flt_Modules[0].27) XIC(Flt_Modules[0].28) XIC(Flt_Modules[0].29) XIC(Flt_Modules[0].30) XIC(Flt_Modules[0].31) ]NOP();
   // ------------ General I/O Module Faults ------------------------------------
   17: MOV(Flt_Modules[0],FltsToCitect[5]);
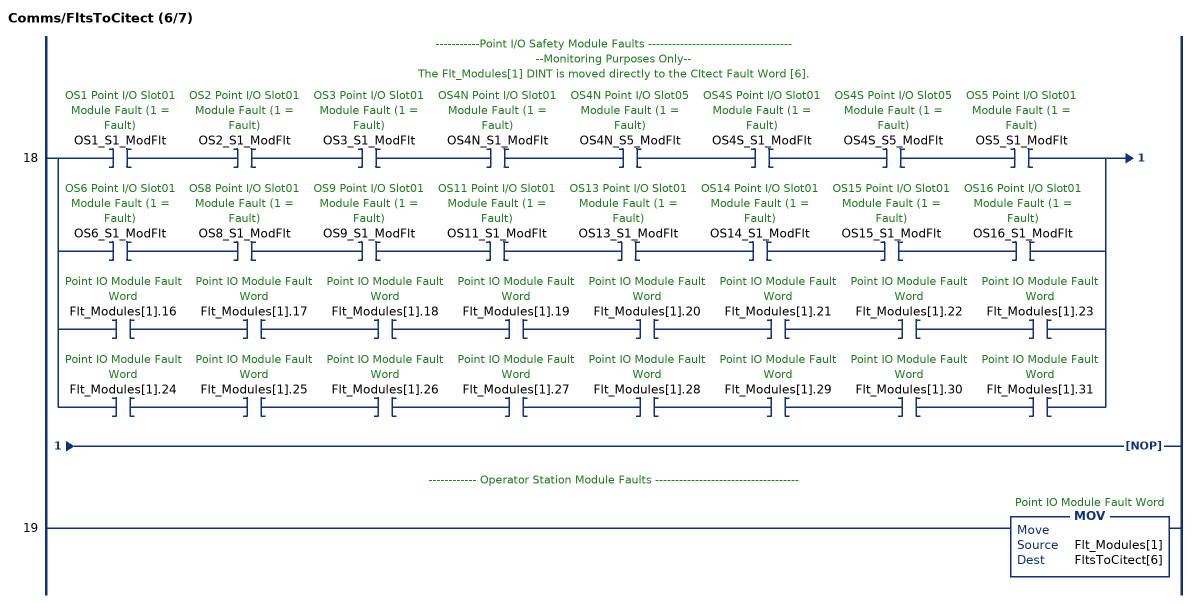
   // -----------Point I/O Safety Module Faults ------------------------------------
   // --Monitoring Purposes Only--
   // The Flt_Modules[1] DINT is moved directly to the CItect Fault Word [6].
   18: [XIC(OS1_S1_ModFlt) XIC(OS2_S1_ModFlt) XIC(OS3_S1_ModFlt) XIC(OS4N_S1_ModFlt) XIC(OS4N_S5_ModFlt) XIC(OS4S_S1_ModFlt) XIC(OS4S_S5_ModFlt) XIC(OS5_S1_ModFlt) ,XIC(OS6_S1_ModFlt) XIC(OS8_S1_ModFlt) XIC(OS9_S1_ModFlt) XIC(OS11_S1_ModFlt) XIC(OS13_S1_ModFlt) XIC(OS14_S1_ModFlt) XIC(OS15_S1_ModFlt) XIC(OS16_S1_ModFlt) ,XIC(Flt_Modules[1].16) XIC(Flt_Modules[1].17) XIC(Flt_Modules[1].18) XIC(Flt_Modules[1].19) XIC(Flt_Modules[1].20) XIC(Flt_Modules[1].21) XIC(Flt_Modules[1].22) XIC(Flt_Modules[1].23) ,XIC(Flt_Modules[1].24) XIC(Flt_Modules[1].25) XIC(Flt_Modules[1].26) XIC(Flt_Modules[1].27) XIC(Flt_Modules[1].28) XIC(Flt_Modules[1].29) XIC(Flt_Modules[1].30) XIC(Flt_Modules[1].31) ]NOP();
   // ------------ Operator Station Module Faults ------------------------------------
   19: MOV(Flt_Modules[1],FltsToCitect[6]);
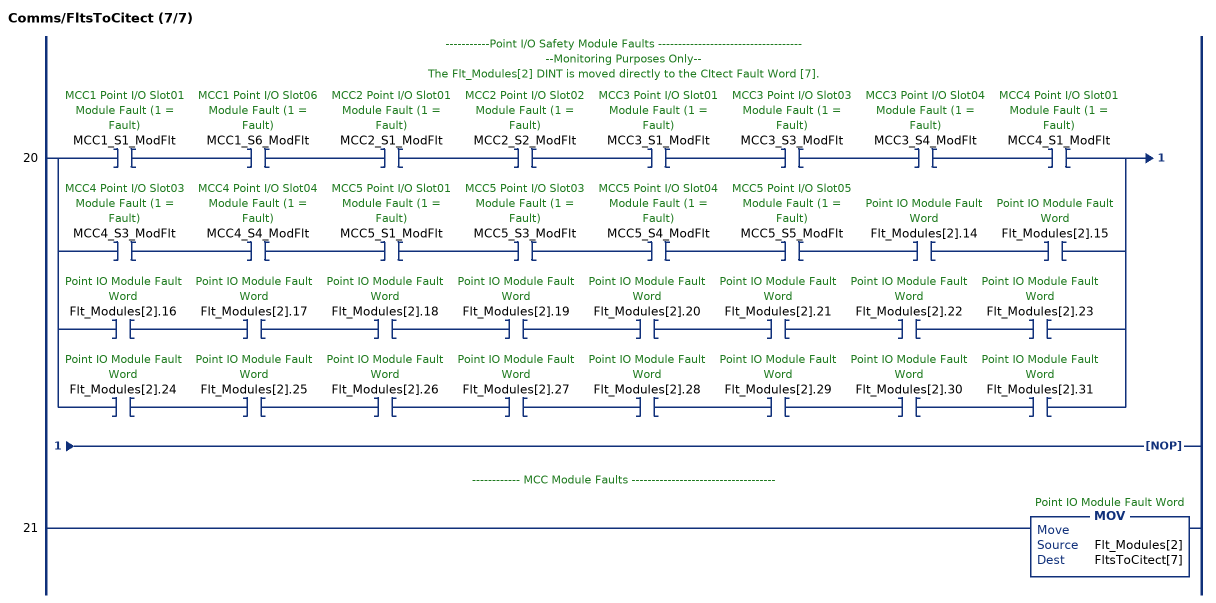
   // -----------Point I/O Safety Module Faults ------------------------------------
   // --Monitoring Purposes Only--
   // The Flt_Modules[2] DINT is moved directly to the CItect Fault Word [7].
   20: [XIC(MCC1_S1_ModFlt) XIC(MCC1_S6_ModFlt) XIC(MCC2_S1_ModFlt) XIC(MCC2_S2_ModFlt) XIC(MCC3_S1_ModFlt) XIC(MCC3_S3_ModFlt) XIC(MCC3_S4_ModFlt) XIC(MCC4_S1_ModFlt) ,XIC(MCC4_S3_ModFlt) XIC(MCC4_S4_ModFlt) XIC(MCC5_S1_ModFlt) XIC(MCC5_S3_ModFlt) XIC(MCC5_S4_ModFlt) XIC(MCC5_S5_ModFlt) XIC(Flt_Modules[2].14) XIC(Flt_Modules[2].15) ,XIC(Flt_Modules[2].16) XIC(Flt_Modules[2].17) XIC(Flt_Modules[2].18) XIC(Flt_Modules[2].19) XIC(Flt_Modules[2].20) XIC(Flt_Modules[2].21) XIC(Flt_Modules[2].22) XIC(Flt_Modules[2].23) ,XIC(Flt_Modules[2].24) XIC(Flt_Modules[2].25) XIC(Flt_Modules[2].26) XIC(Flt_Modules[2].27) XIC(Flt_Modules[2].28) XIC(Flt_Modules[2].29) XIC(Flt_Modules[2].30) XIC(Flt_Modules[2].31) ]NOP();
   // ------------ MCC Module Faults ------------------------------------
   21: MOV(Flt_Modules[2],FltsToCitect[7]);
END_ROUTINE

ROUTINE FromCitect   (* ladder *)
// Signals
// From Citect System
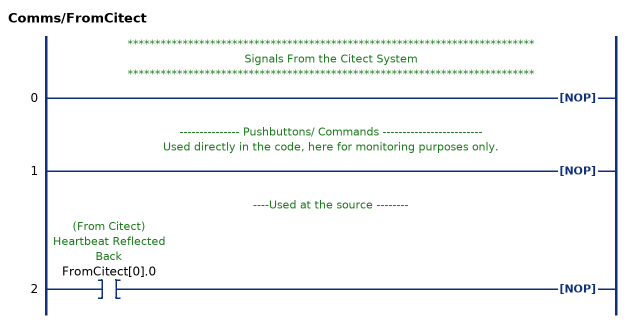
   // **************************************************************************
   // Signals From the Citect System
   // **************************************************************************
   0: NOP();
   // --------------- Pushbuttons/ Commands -------------------------
   // Used directly in the code, here for monitoring purposes only.
   1: NOP();
   // ----Used at the source --------
   2: XIC(FromCitect[0].0)NOP();
END_ROUTINE

ROUTINE FromMach   (* ladder *)
// Signals
// from Machine Processor
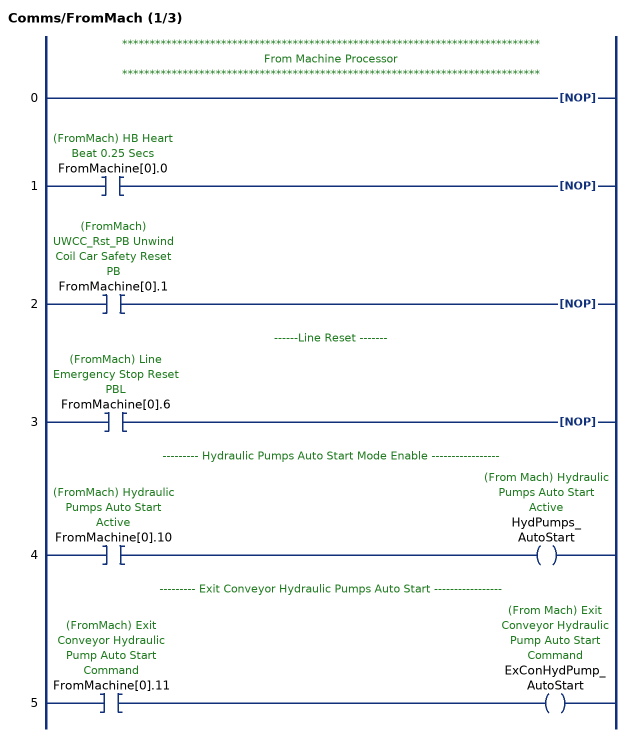
   // ****************************************************************************
   // From Machine Processor
   // ****************************************************************************
   0: NOP();
   1: XIC(FromMachine[0].0)NOP();
   2: XIC(FromMachine[0].1)NOP();
   // ------Line Reset -------
   3: XIC(FromMachine[0].6)NOP();
   // --------- Hydraulic Pumps Auto Start Mode Enable -----------------
   4: XIC(FromMachine[0].10)OTE(HydPumps_AutoStart);
   // --------- Exit Conveyor Hydraulic Pumps Auto Start -----------------
   5: XIC(FromMachine[0].11)OTE(ExConHydPump_AutoStart);
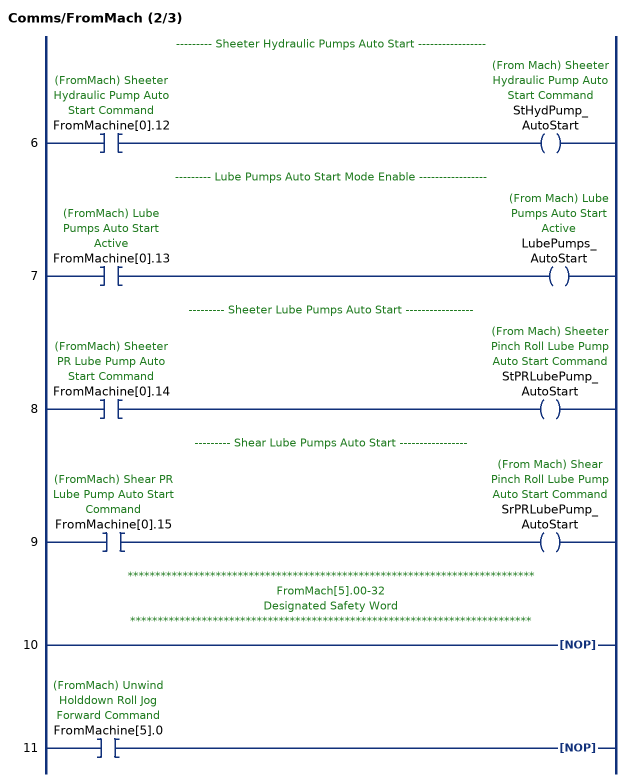
   // --------- Sheeter Hydraulic Pumps Auto Start -----------------
   6: XIC(FromMachine[0].12)OTE(StHydPump_AutoStart);
   // --------- Lube Pumps Auto Start Mode Enable -----------------
   7: XIC(FromMachine[0].13)OTE(LubePumps_AutoStart);
   // --------- Sheeter Lube Pumps Auto Start -----------------
   8: XIC(FromMachine[0].14)OTE(StPRLubePump_AutoStart);
   // --------- Shear Lube Pumps Auto Start -----------------
   9: XIC(FromMachine[0].15)OTE(SrPRLubePump_AutoStart);
   // **************************************************************************
   // FromMach[5].00-32
   // Designated Safety Word
   // *************************************************************************
   10: NOP();
   11: XIC(FromMachine[5].0)NOP();
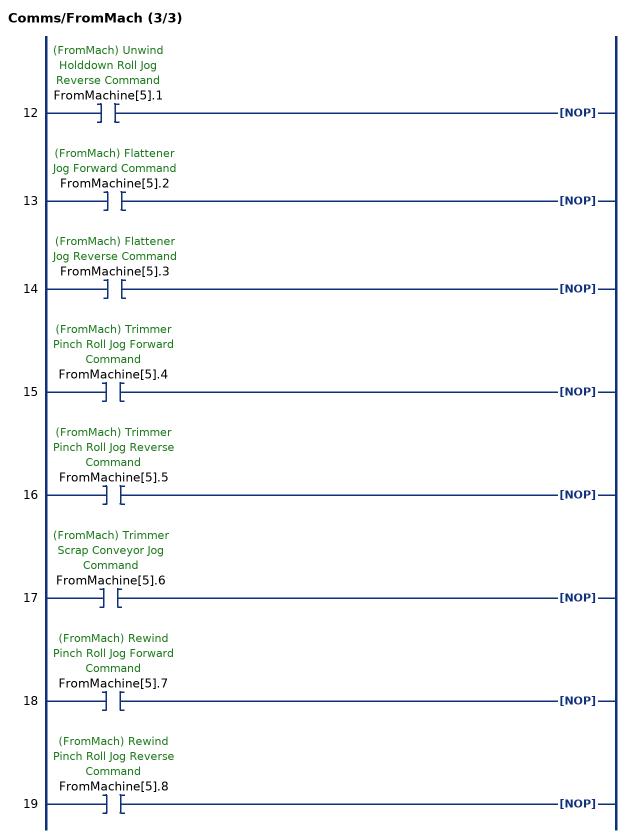
   12: XIC(FromMachine[5].1)NOP();
   13: XIC(FromMachine[5].2)NOP();
   14: XIC(FromMachine[5].3)NOP();
   15: XIC(FromMachine[5].4)NOP();
   16: XIC(FromMachine[5].5)NOP();
   17: XIC(FromMachine[5].6)NOP();
   18: XIC(FromMachine[5].7)NOP();
   19: XIC(FromMachine[5].8)NOP();
END_ROUTINE

ROUTINE FromShDie   (* ladder *)
// Signals
// from Shear Die Processor
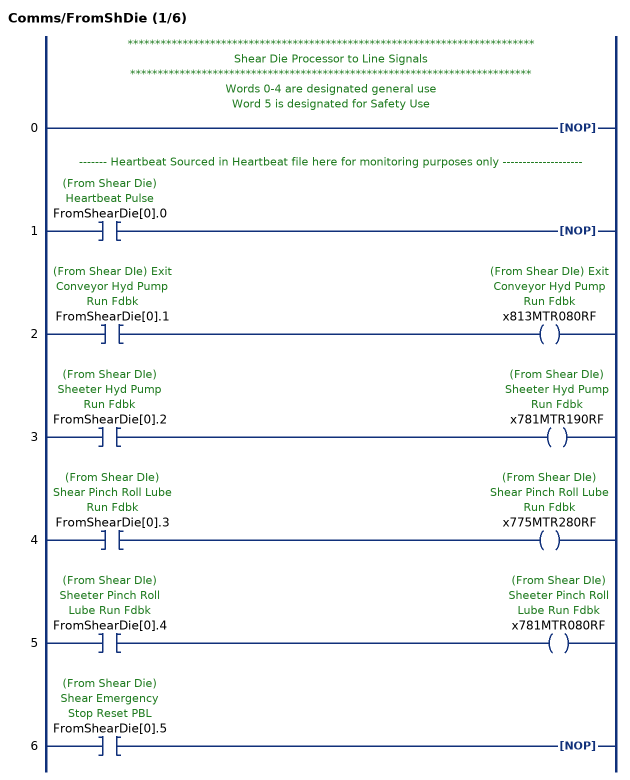
   // **************************************************************************
   // Shear Die Processor to Line Signals
   // *************************************************************************
   // Words 0-4 are designated general use
   // Word 5 is designated for Safety Use
   0: NOP();
   // ------- Heartbeat Sourced in Heartbeat file here for monitoring purposes only --------------------
   1: XIC(FromShearDie[0].0)NOP();
   2: XIC(FromShearDie[0].1)OTE(x813MTR080RF);
   3: XIC(FromShearDie[0].2)OTE(x781MTR190RF);
   4: XIC(FromShearDie[0].3)OTE(x775MTR280RF);
   5: XIC(FromShearDie[0].4)OTE(x781MTR080RF);
   6: XIC(FromShearDie[0].5)NOP();
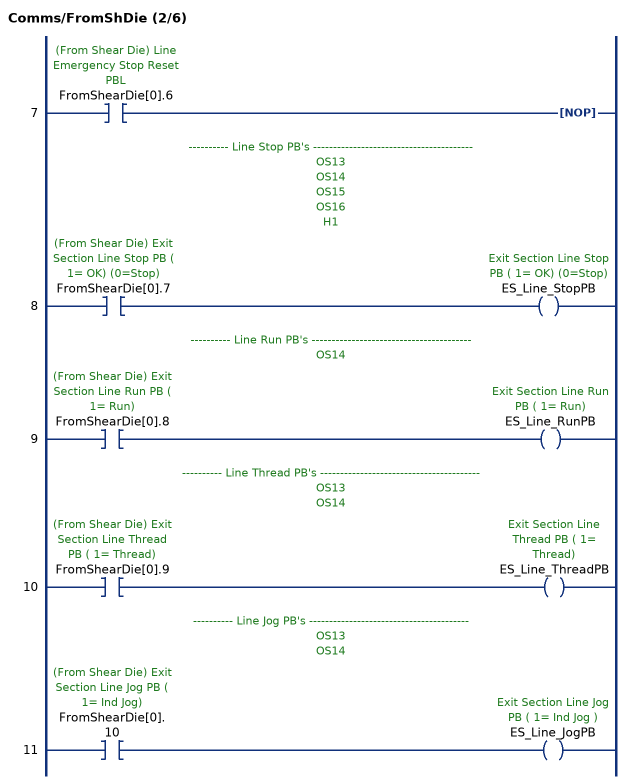
   7: XIC(FromShearDie[0].6)NOP();
   // ---------- Line Stop PB's ----------------------------------------
   // OS13
   // OS14
   // OS15
   // OS16
   // H1
   8: XIC(FromShearDie[0].7)OTE(ES_Line_StopPB);
   // ---------- Line Run PB's ----------------------------------------
   // OS14
   9: XIC(FromShearDie[0].8)OTE(ES_Line_RunPB);
   // ---------- Line Thread PB's ----------------------------------------
   // OS13
   // OS14
   10: XIC(FromShearDie[0].9)OTE(ES_Line_ThreadPB);
   // ---------- Line Jog PB's ----------------------------------------
   // OS13
   // OS14
   11: XIC(FromShearDie[0].10)OTE(ES_Line_JogPB);
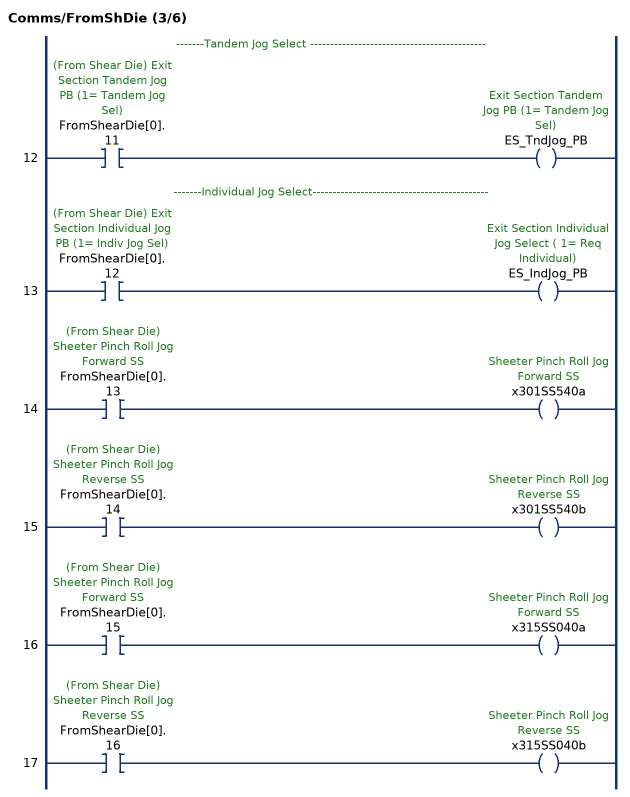
   // -------Tandem Jog Select --------------------------------------------
   12: XIC(FromShearDie[0].11)OTE(ES_TndJog_PB);
   // -------Individual Jog Select--------------------------------------------
   13: XIC(FromShearDie[0].12)OTE(ES_IndJog_PB);
   14: XIC(FromShearDie[0].13)OTE(x301SS540a);
   15: XIC(FromShearDie[0].14)OTE(x301SS540b);
   16: XIC(FromShearDie[0].15)OTE(x315SS040a);
   17: XIC(FromShearDie[0].16)OTE(x315SS040b);
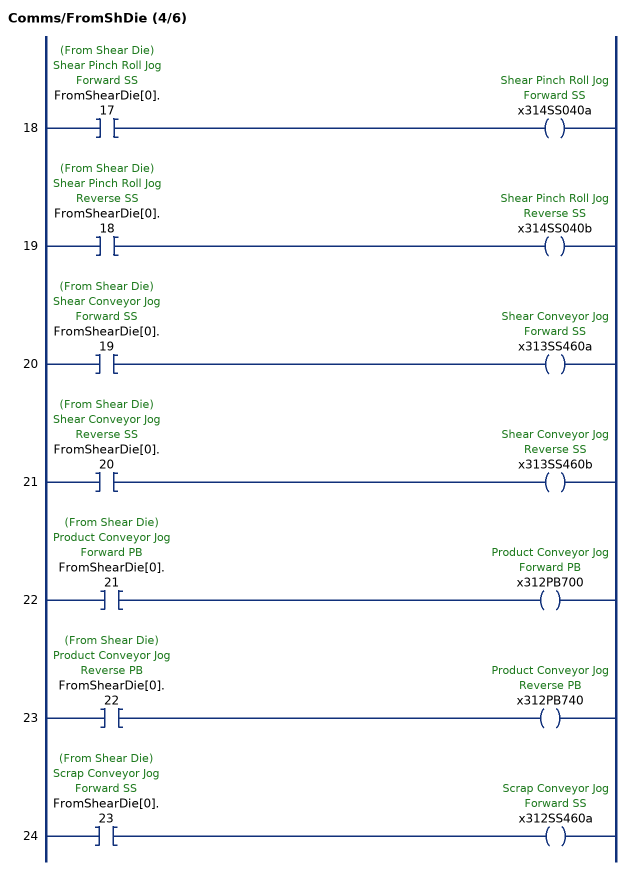
   18: XIC(FromShearDie[0].17)OTE(x314SS040a);
   19: XIC(FromShearDie[0].18)OTE(x314SS040b);
   20: XIC(FromShearDie[0].19)OTE(x313SS460a);
   21: XIC(FromShearDie[0].20)OTE(x313SS460b);
   22: XIC(FromShearDie[0].21)OTE(x312PB700);
   23: XIC(FromShearDie[0].22)OTE(x312PB740);
   24: XIC(FromShearDie[0].23)OTE(x312SS460a);
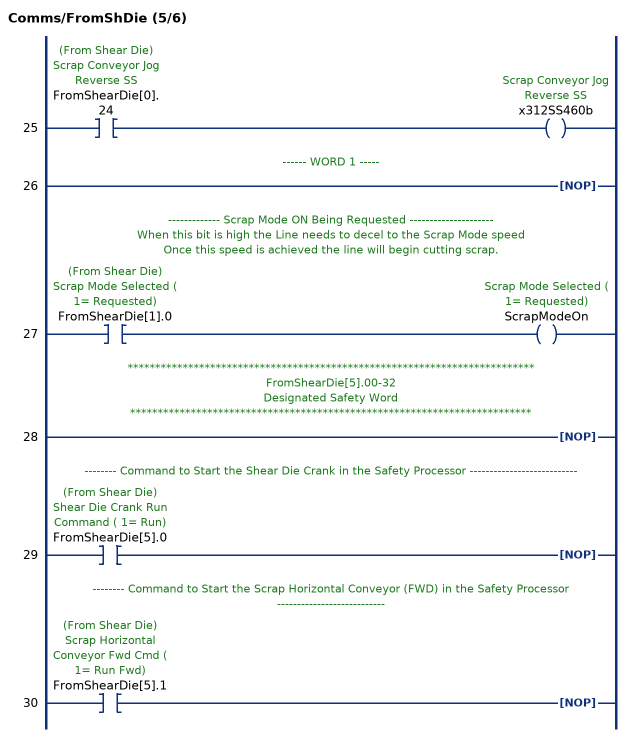
   25: XIC(FromShearDie[0].24)OTE(x312SS460b);
   // ------ WORD 1 -----
   26: NOP();
   // ------------- Scrap Mode ON Being Requested ---------------------
   // When this bit is high the Line needs to decel to the Scrap Mode speed
   // Once this speed is achieved the line will begin cutting scrap.
   27: XIC(FromShearDie[1].0)OTE(ScrapModeOn);
   // **************************************************************************
   // FromShearDie[5].00-32
   // Designated Safety Word
   // *************************************************************************
   28: NOP();
   // -------- Command to Start the Shear Die Crank in the Safety Processor ---------------------------
   29: XIC(FromShearDie[5].0)NOP();
   // -------- Command to Start the Scrap Horizontal Conveyor (FWD) in the Safety Processor ---------------------------
   30: XIC(FromShearDie[5].1)NOP();
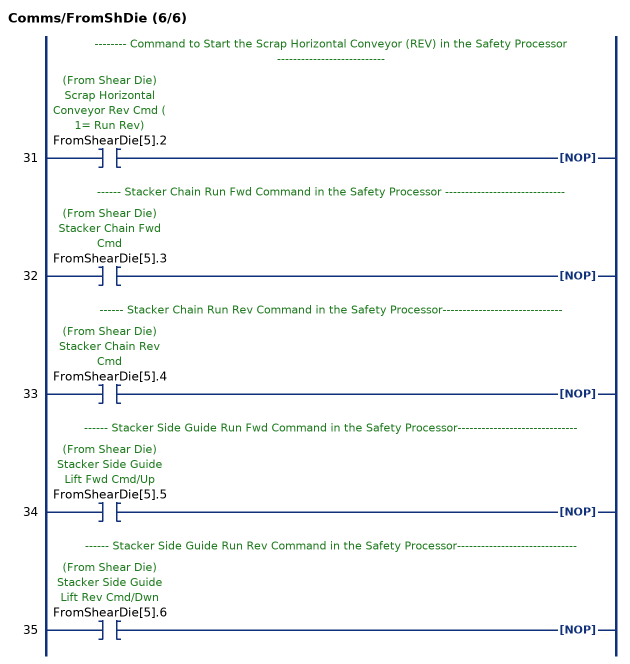
   // -------- Command to Start the Scrap Horizontal Conveyor (REV) in the Safety Processor ---------------------------
   31: XIC(FromShearDie[5].2)NOP();
   // ------ Stacker Chain Run Fwd Command in the Safety Processor ------------------------------
   32: XIC(FromShearDie[5].3)NOP();
   // ------ Stacker Chain Run Rev Command in the Safety Processor------------------------------
   33: XIC(FromShearDie[5].4)NOP();
   // ------ Stacker Side Guide Run Fwd Command in the Safety Processor------------------------------
   34: XIC(FromShearDie[5].5)NOP();
   // ------ Stacker Side Guide Run Rev Command in the Safety Processor------------------------------
   35: XIC(FromShearDie[5].6)NOP();
END_ROUTINE
